// TIA Portal V20 export
DATA_BLOCK "PM01"   // DB334
// stored: MemoryReserve 100
   VAR
      "SEPA DANCER FORWARD" : Bool := FALSE;
      "SEPA DANCER BACKWARD" : Bool := FALSE;
      "SEPA UW #1 IONIZER TOP ON" : Bool := FALSE;
      SPARE : Bool := FALSE;
      "SEPA UW #1 IONIZER BTM ON" : Bool := FALSE;
      SPARE_1 : Bool := FALSE;
      "SEPA UW #1 AIR SHAFT TOP ON" : Bool := FALSE;
      "SEPA UW #1 AIR SHAFT TOP OFF" : Bool := FALSE;
      "SEPA UW #1 AIR SHAFT BTM ON" : Bool := FALSE;
      "SEPA UW #1 AIR SHAFT BTM OFF" : Bool := FALSE;
      SPARE_3 : Bool := FALSE;
      SPARE_4 : Bool := FALSE;
      "ANODE CONVEYOR PICK UP BLOWER ON/OFF" : Bool := FALSE;
      SPARE_2 : Bool := FALSE;
      "CATHODE CONVEYOR PICK UP BLOWER ON/OFF" : Bool := FALSE;
   END_VAR
BEGIN
END_DATA_BLOCK
